INTERFACE INullReferenceException EXTENDS IGeneralException

METHOD Throw
VAR_INPUT
	sourceNamespaceName : STRING;
	sourceClassName : STRING;
	sourcePOUName : STRING;
	sourcePosition : STRING;
	variableOrPropertyName : STRING;
END_VAR
END_METHOD

END_INTERFACE

(* stored: Version 1.1.0.1
   Itf INullReferenceException: Id {038e712d-4ef6-48ba-830c-6ff3d9907d05}
   Method Throw: Id {c610b497-8802-47d6-934b-8a411e820c9b} *)
